Yaskawa INFORM job: PURGE.JBI

/JOB
//NAME PURGE
//POS
///NPOS 0,0,0,0,0,0
//INST
///DATE 2018/09/25 14:14
///ATTR SC,RW,MC
///LVARS 5,5,0,0,0,0,0,0
NOP
GETARG LB000 IARG#(1)
SET LI000 LB000
MUL LI000 100
PULSE OT#(25) T=LI000
TIMER T=LI000
END
